PROGRAM ManualDosingSTreset
VAR

END_VAR

(*Function to reset the manual button in Recipe Mode*)(*Changes On 12/12/17-Andy*)
(*Additional Input For Dosing enable function-Add bStn1ManualDosingST*)(*Changes On 12/12/17-Andy*)

IF NOT ManualPageEnable THEN

	IF ARbStnManualDosingDone[1] THEN

		ARbStnManualDosingST[1] :=FALSE;

	ELSIF ARbStnManualDosingDone[3] THEN

		ARbStnManualDosingST[3] :=FALSE;
		
	ELSIF ARbStnManualDosingDone[5] THEN

		ARbStnManualDosingST[5] :=FALSE;
	END_IF

END_IF

END_PROGRAM

(* stored: Version 1.1.0.1, ProductVersion 3.1.4024.12
   POU ManualDosingSTreset: Id {b5b79887-a37a-42cb-b728-35745c8d3e88}, SpecialFunc None *)
